# EPICS autosave request: BPMApp/Db/BPMIntlk_settings.req
$(P)$(R)IntlkEn-Sel
$(P)$(R)IntlkMinSumEn-Sel
$(P)$(R)IntlkTransEn-Sel
$(P)$(R)IntlkAngEn-Sel
$(P)$(R)IntlkLmtMinSum-SP
$(P)$(R)IntlkLmtTransMaxX-SP
$(P)$(R)IntlkLmtTransMaxY-SP
$(P)$(R)IntlkLmtAngMaxX-SP
$(P)$(R)IntlkLmtAngMaxY-SP
